// TIA Portal V17 export
// export: Created 2024-09-02T12:49:54.5362234Z, ExportSetting WithDefaults, DisplayName Totally Integrated Automation Portal, DisplayVersion V17, DisplayName TIA Portal Openness, DisplayVersion V17, DisplayName TIA Portal Version Control Interface, DisplayVersion V17, DisplayName STEP 7 Professional, DisplayVersion V17, DisplayName STEP 7 Safety, DisplayVersion V17, DisplayName WinCC Professional, DisplayVersion V17
ORGANIZATION_BLOCK "MainAnwender"   // OB1001, LAD, ProgramCycle
TITLE = "Main Program Sweep (Cycle)"
{ S7_Optimized_Access := 'TRUE' }
AUTHOR : OlegFuehrus
VERSION : 0.1
// stored: AutoNumber false, IsIECCheckEnabled false, SetENOAutomatically false
   VAR_INPUT
      Initial_Call : Bool;   // Initial call of this OB
      Remanence : Bool;   // =True, if remanent data are available
   END_VAR
   VAR_TEMP
      retVal : Word;
      leftFunction : Bool;
      rightFunction : Bool;
      scaleNumberOK : Bool;
      errID : Word;
      t_ret : Word;
      t_Anz : Int;
      t_Fehler : Bool;
      t_Funktion_links : Bool;
      t_Funktion_rechts : Bool;
   END_VAR
BEGIN

REGION Network 1: HandMovement Refreshing
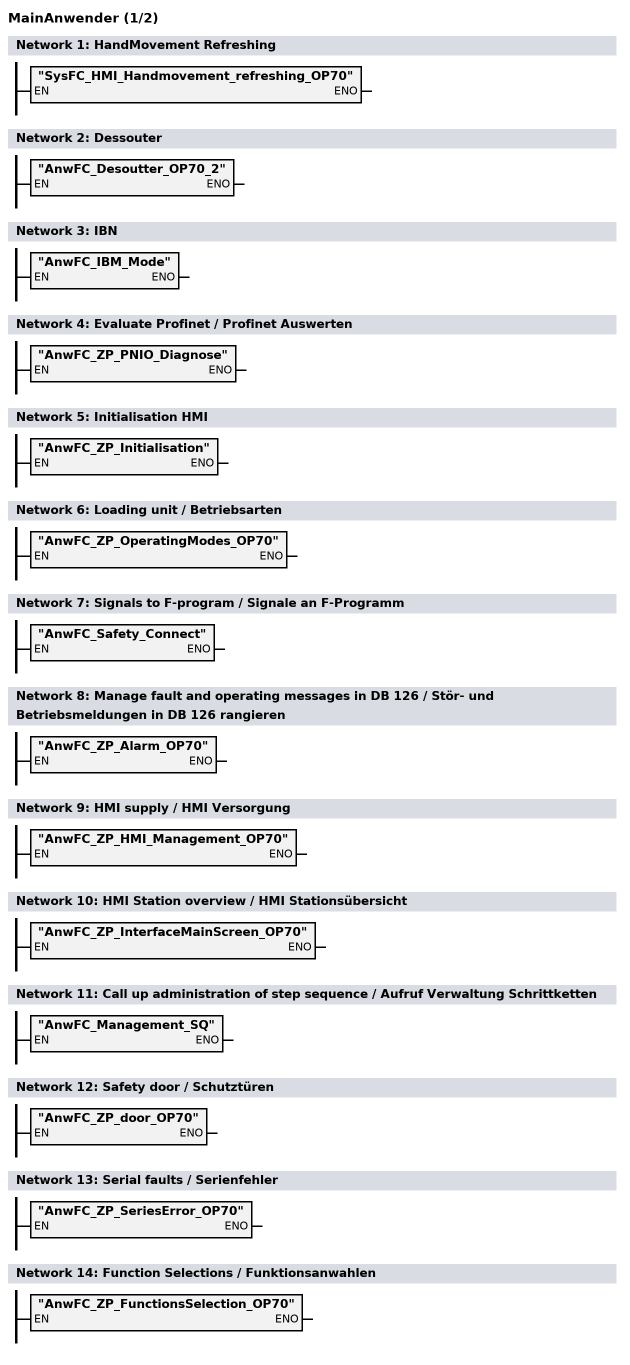
   RUNG wire#powerrail
      "SysFC_HMI_Handmovement_refreshing_OP70"()
   END_RUNG
   // the same network as SCL:
   "SysFC_HMI_Handmovement_refreshing_OP70"();
END_REGION

REGION Network 2: Dessouter
   RUNG wire#powerrail
      "AnwFC_Desoutter_OP70_2"()
   END_RUNG
   // the same network as SCL:
   "AnwFC_Desoutter_OP70_2"();
END_REGION

REGION Network 3: IBN
   RUNG wire#powerrail
      "AnwFC_IBM_Mode"()
   END_RUNG
   // the same network as SCL:
   "AnwFC_IBM_Mode"();
END_REGION

REGION Network 4: Evaluate Profinet / Profinet Auswerten
   RUNG wire#powerrail
      "AnwFC_ZP_PNIO_Diagnose"()
   END_RUNG
   // the same network as SCL:
   "AnwFC_ZP_PNIO_Diagnose"();
END_REGION

REGION Network 5: Initialisation HMI
   RUNG wire#powerrail
      "AnwFC_ZP_Initialisation"()
   END_RUNG
   // the same network as SCL:
   "AnwFC_ZP_Initialisation"();
END_REGION

REGION Network 6: Loading unit / Betriebsarten
   RUNG wire#powerrail
      "AnwFC_ZP_OperatingModes_OP70"()
   END_RUNG
   // the same network as SCL:
   "AnwFC_ZP_OperatingModes_OP70"();
END_REGION

REGION Network 7: Signals to F-program / Signale an F-Programm
   RUNG wire#powerrail
      "AnwFC_Safety_Connect"()
   END_RUNG
   // the same network as SCL:
   "AnwFC_Safety_Connect"();
END_REGION

REGION Network 8: Manage fault and operating messages in DB 126 / Stör- und Betriebsmeldungen in DB 126 rangieren
   RUNG wire#powerrail
      "AnwFC_ZP_Alarm_OP70"()
   END_RUNG
   // the same network as SCL:
   "AnwFC_ZP_Alarm_OP70"();
END_REGION

REGION Network 9: HMI supply / HMI Versorgung
   RUNG wire#powerrail
      "AnwFC_ZP_HMI_Management_OP70"()
   END_RUNG
   // the same network as SCL:
   "AnwFC_ZP_HMI_Management_OP70"();
END_REGION

REGION Network 10: HMI Station overview / HMI Stationsübersicht
   RUNG wire#powerrail
      "AnwFC_ZP_InterfaceMainScreen_OP70"()
   END_RUNG
   // the same network as SCL:
   "AnwFC_ZP_InterfaceMainScreen_OP70"();
END_REGION

REGION Network 11: Call up administration of step sequence / Aufruf Verwaltung Schrittketten
   RUNG wire#powerrail
      "AnwFC_Management_SQ"()
   END_RUNG
   // the same network as SCL:
   "AnwFC_Management_SQ"();
END_REGION

REGION Network 12: Safety door / Schutztüren
   RUNG wire#powerrail
      "AnwFC_ZP_door_OP70"()
   END_RUNG
   // the same network as SCL:
   "AnwFC_ZP_door_OP70"();
END_REGION

REGION Network 13: Serial faults / Serienfehler
   RUNG wire#powerrail
      "AnwFC_ZP_SeriesError_OP70"()
   END_RUNG
   // the same network as SCL:
   "AnwFC_ZP_SeriesError_OP70"();
END_REGION

REGION Network 14: Function Selections / Funktionsanwahlen
   RUNG wire#powerrail
      "AnwFC_ZP_FunctionsSelection_OP70"()
   END_RUNG
   // the same network as SCL:
   "AnwFC_ZP_FunctionsSelection_OP70"();
END_REGION

REGION Network 15: MES
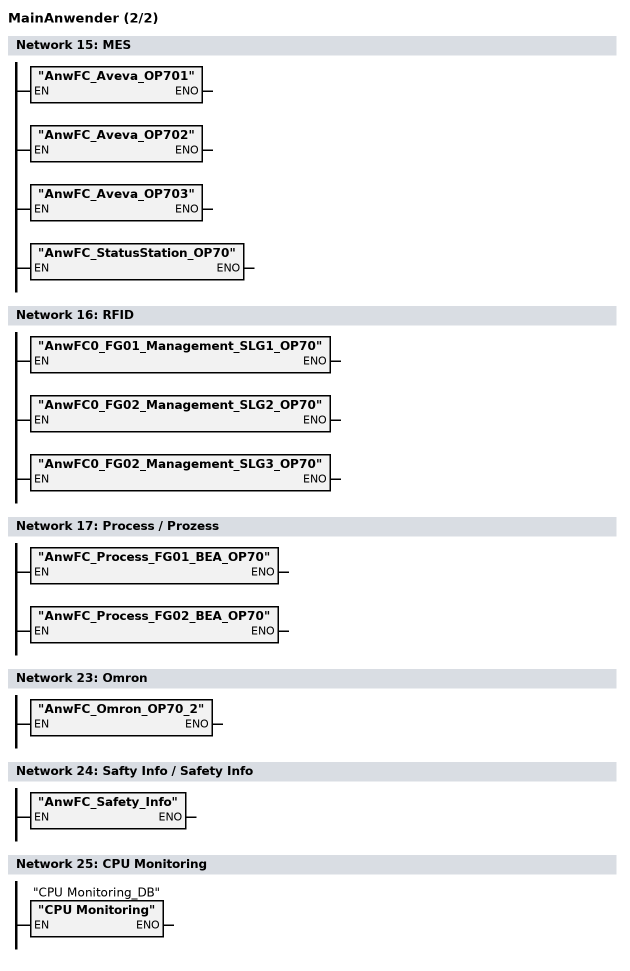
   RUNG wire#powerrail
      "AnwFC_Aveva_OP701"()
   END_RUNG
   RUNG wire#powerrail
      "AnwFC_Aveva_OP702"()
   END_RUNG
   RUNG wire#powerrail
      "AnwFC_Aveva_OP703"()
   END_RUNG
   RUNG wire#powerrail
      "AnwFC_StatusStation_OP70"()
   END_RUNG
   // the same network as SCL:
   "AnwFC_Aveva_OP701"();
   "AnwFC_Aveva_OP702"();
   "AnwFC_Aveva_OP703"();
   "AnwFC_StatusStation_OP70"();
END_REGION

REGION Network 16: RFID
   RUNG wire#powerrail
      "AnwFC0_FG01_Management_SLG1_OP70"()
   END_RUNG
   RUNG wire#powerrail
      "AnwFC0_FG02_Management_SLG2_OP70"()
   END_RUNG
   RUNG wire#powerrail
      "AnwFC0_FG02_Management_SLG3_OP70"()
   END_RUNG
   // the same network as SCL:
   "AnwFC0_FG01_Management_SLG1_OP70"();
   "AnwFC0_FG02_Management_SLG2_OP70"();
   "AnwFC0_FG02_Management_SLG3_OP70"();
END_REGION

REGION Network 17: Process / Prozess
   RUNG wire#powerrail
      "AnwFC_Process_FG01_BEA_OP70"()
   END_RUNG
   RUNG wire#powerrail
      "AnwFC_Process_FG02_BEA_OP70"()
   END_RUNG
   // the same network as SCL:
   "AnwFC_Process_FG01_BEA_OP70"();
   "AnwFC_Process_FG02_BEA_OP70"();
END_REGION

REGION Network 18: Sinamics S120
END_REGION

REGION Network 19: MPRO
END_REGION

REGION Network 20: maXYmos
END_REGION

REGION Network 21: Ehternet
END_REGION

REGION Network 22: Lubrication / Schmierung
END_REGION

REGION Network 23: Omron
   RUNG wire#powerrail
      "AnwFC_Omron_OP70_2"()
   END_RUNG
   // the same network as SCL:
   "AnwFC_Omron_OP70_2"();
END_REGION

REGION Network 24: Safty Info / Safety Info
   RUNG wire#powerrail
      "AnwFC_Safety_Info"()
   END_RUNG
   // the same network as SCL:
   "AnwFC_Safety_Info"();
END_REGION

REGION Network 25: CPU Monitoring
   RUNG wire#powerrail
      "CPU Monitoring_DB"()
   END_RUNG
   // the same network as SCL:
   "CPU Monitoring_DB"();   // "CPU Monitoring"
END_REGION
END_ORGANIZATION_BLOCK
